(* CODESYS project festo_cpx_api_ec_beckhoff.library
   DefaultNamespace: Festo_CPX_AP_I_EC
   DocFormat: reStructuredText
   Description: FB's for integrating CPX_AP_I_EC_M12 module
   Author: INOSKSR
   Title: Festo_CPX_API_EC_Beckhoff
   Version: 3.5.12.2
   Company: Festo
   Placeholder: Festo_CPX_AP_I_EC

Project tree, tasks and I/O mapping:
  libraries: Tc2_EtherCAT, * (Beckhoff Automation GmbH); Tc2_Standard, * (Beckhoff Automation GmbH); Tc2_System, * (Beckhoff Automation GmbH); Tc3_Module, * (Beckhoff Automation GmbH)
  DUTs/
    function block Restart_Slave [ST]
    data type stModuleDiagData
  ENUMs/
    data type eErrorDescription
    data type eIOLinkAbortCode
    data type eSDOAbortCode
  POUs/
    function block CPXAPI_Diag [ST]
    function block CPXAPI_IOLink_Parameter [ST]
    function block CPXAPI_Parameter [ST]
  Project Information/
    function F_GetCompany [ST]
    function F_GetTitle [ST]
    function F_GetVersion [ST]
  UNIONs/
    data type UDINT_AS_ARRAYOFBYTE
    data type UINT_AS_ARRAYOFBYTE
  Version/
    global variables Global_Version
  VISUs/
    visualisation VISU_CPXAPI_Diag
    visualisation VISU_CPXAPI_IOLinkParameter
    visualisation VISU_CPXAPI_Parameter
  text list GlobalTextList
*)

// DUTs/stModuleDiagData
TYPE stModuleDiagData :
STRUCT
	udiModuleDiagState     : UDINT;
    uiActiveDiagnosisCount : UINT;
	uiSubModule            : UINT;
	uiChannel              : UINT;
	udiDiagnosisCode       : UDINT;
	eErrorDescription      : eErrorDescription;
	xError                 : BOOL;
END_STRUCT
END_TYPE

// ENUMs/eErrorDescription
TYPE eErrorDescription :
(
	NO_ERROR                                              := 0 ,
	OVERVOLTAGE_LOAD_SUPPLY_PS                            := 33619991,
	UNDERVOLTAGE_LOAD_SUPPLY_PL                           := 33620229,
	SWITCH_OFF_LOAD_SUPPLY_PL                             := 33620230,
	OVERVOLTAGE_LOAD_SUPPLY_PL                            := 33620287,
	START_UP_PARAMETER_REJECTED                           := 100663561,
	START_UP_PARAMETER_DEVIATION_IN_LENGTH                := 100663562,
	MODULE_IDENTIFICATION_CHECK_SKIPPED                   := 100663688,
	MODULE_IDENTIFICATION_CHECK_FAILED                    := 100663689,
	DEVICE_ADDRESS_INVALID                                := 134218030,
	INVALID_CYCLE_TIME                                    := 134218130,
	AP_MASTER_LOST                                        := 134283556,
	COMMUNICATION_TO_AP_MODULE_INTERRUPTED                := 134283559,
	OUTPUT_PROCESS_DATA_WATCHDOG_OF_THE_AP_MODULE_EXPIRED := 134283568,
	INPUT_PROCESS_DATA_WATCHDOG_OF_THE_AP_MODULE_EXPIRED  := 134283569,                                   
	OUTPUT_PROCESS_DATA_WATCHDOG_OF_THE_INTERFACE_EXPIRED := 134283570,
	INPUT_PROCESS_DATA_WATCHDOG_OF_THE_INTERFACE_EXPIRED  := 134283571,	
	AP_MASTER_TOGGLE_BIT_ERROR                            := 134283572,
	STATUS_CHANGE_REQUEST                                 := 134480273,
	SYNC_MANAGER_INVALID_ADDRESS                          := 134480275,
	SYNC_MANAGER_INVALID_IO_SIZE                          := 134480276,
	SYNC_MANAGER_INVALID_CONFIGURATION                    := 134480277,
	DC_ACTIVATION_REGISTER_INVALID                        := 134480278,
	SYNC_TYPE_NOT_SUPPORTED                               := 134480279,
	SYSTEM_START                                          := 184549696,
	FIRMWARE_INVALID                                      := 184811703,
	UNSUPPORTED_FULL_DIAGNOSTIC_IMAGE_VERSION             := 185074063,
	UNSUPPORTED_DIAGNOSTIC_VERSION                        := 185074064,
	APDD_INVALID                                          := 185139496,
	START_UP_APDD_INVALID                                 := 185139497,
	INVALID_SLAVEID_OR_COMMUNICATION_ERROR                := 65535
)DWORD;
END_TYPE

// ENUMs/eIOLinkAbortCode
TYPE eIOLinkAbortCode :
(
  NO_ERROR                     := 16#0,
  SERVICE_NOT_AVAILABLE        := 16#8020,
  INDEX_NOT_AVAILABLE          := 16#8011,
  SUB_INDEX_NOT_AVAILABLE      := 16#8012,
  INDEX_NOT_WRITEABLE          := 16#8023 ,
  PARAMETER_VALUE_OUT_OF_RANGE := 16#8030,
  PARAMETER_VALUE_ABOVE_LIMIT  := 16#8031,
  PARAMETER_VALUE_BELOW_LIMIT  := 16#8032,
  PARAMETER_LENGTH_OVERRUN     := 16#8033,
  PARAMETER_LENGTH_UNDERRUN    := 16#8034,
  VENDOR_SPECIFIC              := 16#8181,
  WRONG_SLOT_NUMBER            := 16#703
)DINT;
END_TYPE

// ENUMs/eSDOAbortCode
TYPE eSDOAbortCode :
(
    NO_ERROR                            := 16#0,
	INTERNAL_ERROR                      := 16#1 ,
    NO_REAL_TIME_ERROR                  := 16#2 ,
	PORT_NOT_CONNECTED                  := 16#D,
    GENERAL_DEVICE_ERROR                := 16#700 ,
	SERVICE_NOT_SUPPORTED_BY_SERVER     := 16#701 ,
	INVALID_INDEX_GROUP                 := 16#702 ,
	INVALID_INDEX_OFFSET                := 16#703 , 
	READING_OR_WRITTING_NOT_PERMITTED   := 16#704,
	PARAMETER_SIZE_INCORRECT            := 16#705,
	INVALID_DATA_VALUES                 := 16#706,
	DEVICE_NOT_READY                    := 16#707,
	DEVICE_BUSY                         := 16#708,
	INSUFFICIENT_MEMORY                 := 16#70A,
	INVALID_PARAMETER_VALUES            := 16#70B,
	SYNTAX_ERROR                        := 16#70D
	
	
)DINT;
END_TYPE

// UNIONs/UDINT_AS_ARRAYOFBYTE
TYPE UDINT_AS_ARRAYOFBYTE :
UNION
	dataUDINT: UDINT;
	dataArray : ARRAY[1..4] OF BYTE;
END_UNION
END_TYPE

// UNIONs/UINT_AS_ARRAYOFBYTE
TYPE UINT_AS_ARRAYOFBYTE :
UNION
	dataUINT  : UINT;
	dataArray : ARRAY[1..2] OF BYTE;
END_UNION
END_TYPE

// Version/Global_Version
{attribute 'TcGenerated'}
{attribute 'no-analysis'}
{attribute 'linkalways'}
// This function has been automatically generated from the project information.
VAR_GLOBAL CONSTANT
	{attribute 'const_non_replaced'}
	stLibVersion_Festo_CPX_API_EC_Beckhoff : ST_LibVersion := (iMajor := 3, iMinor := 5, iBuild := 12, iRevision := 2, nFlags := 0, sVersion := '3.5.12.2');
END_VAR

// DUTs/Restart_Slave
FUNCTION_BLOCK Restart_Slave
VAR_INPUT
	xExecute	: 	BOOL;
	sNetId		: 	STRING;
	nSlaveAddr	: 	UINT;
END_VAR
VAR_OUTPUT
	xDone			:	 BOOL;
	xBusy			: 	BOOL;
	xError			: 	BOOL;
	udiError		: 	UDINT;
	stSlaveState	:	Tc2_EtherCAT.ST_EcSlaveState;
END_VAR
VAR
	SetState		: 	FB_EcSetSlaveState;
	GetState		: 	FB_EcGetSlaveState;
	rTrigStart		: 	R_TRIG;
	iStep			: 	INT;
	ReadState		: 	Tc2_EtherCAT.ST_EcSlaveState;
	ExpectedState	: 	UINT := 1;
END_VAR

SetState(sNetId:= sNetId,nSlaveAddr:=nSlaveAddr,tTimeout := T#1S);
GetState(sNetId:= sNetId,nSlaveAddr:=nSlaveAddr,tTimeout := T#1S,state => ReadState);
rTrigStart(CLK := xExecute);

CASE iStep OF
0:
	SetState.bExecute := FALSE;
	GetState.bExecute := FALSE;
	IF rTrigStart.Q THEN
		xBusy := TRUE;
		xError := FALSE;
		xDone := FALSE;
		udiError := 0;
		SetState.reqState := 1;
		ExpectedState := 1;
		iStep := iStep +10;
	END_IF;
	
10:
	SetState.bExecute := TRUE;
	iStep := iStep +10;

20:
	IF NOT SetState.bBusy AND NOT SetState.bError THEN
		SetState.bExecute := FALSE;
		iStep := iStep +10;	
	ELSIF SetState.bError THEN
		udiError := SetState.nErrId;
		iStep := 999;
	END_IF;
	
30:
	GetState.bExecute := TRUE;
	iStep := iStep +10;

40:
	IF NOT GetState.bBusy AND NOT GetState.bError THEN
		GetState.bExecute := FALSE;	
		iStep := iStep +10;
	ELSIF SetState.bError THEN
		udiError := GetState.nErrId;
		iStep := 999;	
	END_IF;
	
50:
	IF ReadState.deviceState = ExpectedState THEN
		SetState.reqState := SHL(SetState.reqState,1);
		ExpectedState := SetState.reqState;
		IF ExpectedState > 8 THEN
			iStep := iStep+10;
		ELSE
			iStep := 10;
		END_IF;
	ELSE
		iStep := 30;
	END_IF;	

60:	
	xBusy := FALSE;
	xError := FALSE;
	xDone := TRUE;
	stSlaveState := ReadState;
	iStep := 0;

999:
	xBusy := FALSE;
	xError := TRUE;
	xDone := FALSE;
	iStep := 0;
	
END_CASE;

END_FUNCTION_BLOCK

// POUs/CPXAPI_Diag
FUNCTION_BLOCK CPXAPI_Diag
VAR_INPUT
	xEnable             : BOOL;              (* TRUE = Start diagnosis continously *)
	sNetId              : STRING;
	uiEthercatAddress   : UINT;              (* Address of the slave device i.e. CPX-AP-I-EC-M12 Module*)
	xRestart            : BOOL;              (* Change Machine State in order INIT, PREOP, SAFE and OPERATIONAL*)
END_VAR

VAR_OUTPUT
	xActive						 : BOOL;	 (*  Diagnosis FB Active *)
	xError                       : BOOL;     (*  Error exists during diagnosis *)
	uiActiveModules              : UINT;     (*  Number of Active modules connected to CPX-AP-I-EC-M12*)
	uiNumberOfActiveErrors       : UINT;     (* Number of Modules with active errors*)
	uiModuleNo                   : UINT;     (* Module with latest diagnostics*)
	aModuleDiagnosticData        : ARRAY[1..150] OF stModuleDiagData ;
END_VAR
VAR
	ReadModuleCount			:	FB_EcCoESdoReadEx;
	ModuleDiagnosis			:	FB_EcCoESdoReadEx;
	aModuleCount			:	ARRAY[1..150] OF UDINT;
	ModuleDiagnosisData		:	ARRAY[1..150] OF BYTE;
	R_Trig_Exec         	:	R_TRIG;
	F_Trig_Exec				:	F_TRIG;
	iStep					:	INT;
	Delay					:	TON;
	xDelay					:	BOOL;
	DelayUpdate				:	TON;
	xDelayUpdate			:	BOOL;
	i						:	INT;
	k						:	INT;
	Acknowledge_Trig		:	R_TRIG;
	Restart_RTrig         	:	R_TRIG;
	iRestart				:	INT;
	Restart_FTrig			:	F_TRIG;
	diActualIndex         	:	DINT;
	iCurrentModuleDiag    	: 	INT;
	DiagCode				:	DWORD;
	ModuleDiagState			:	UDINT_AS_ARRAYOFBYTE;
	DiagnosisCode			:	UDINT_AS_ARRAYOFBYTE;
	SubModule				: 	UINT_AS_ARRAYOFBYTE;
	Channel					: 	UINT_AS_ARRAYOFBYTE;
	NumberOfActiveModules	: 	UINT_AS_ARRAYOFBYTE;
	j                     	: 	INT;
	l                     	: 	INT;
	tempmodules           	: 	ARRAY[1..150] OF INT;
	DelayRequestSlave		:	TON;
	xDelayRequestSlave		:	BOOL;
	iActive					:	INT;
	F_Trig_Active			:	F_TRIG;
	ActiveOff				:	TON;
	xActiveOff				:	BOOL;
	DelayON					:	TON;
	xDelayON				:	BOOL;
	iRestartCount			:	INT;
	iCurrentRestartCount	:	INT;
	SlaveChangeState		: 	Restart_Slave;
	GetSlaveState			:	FB_EcGetSlaveState;
END_VAR

R_Trig_Exec( CLK := xEnable);
F_Trig_Exec( CLK := xEnable);
Restart_RTrig( CLK := xRestart);
Restart_FTrig( CLK := xRestart);
F_Trig_Active( CLK := xActive);

Delay ( IN := xDelay, PT:= T#100MS);
DelayUpdate ( IN := xDelayUpdate, PT:= T#50MS);

ActiveOff ( IN := xActiveOff, PT:= T#500MS);

DelayON ( IN := xDelayON, PT := T#1S );

DelayRequestSlave ( IN := xDelayRequestSlave, PT:= T#50MS);

IF Restart_RTrig.Q THEN
	iRestartCount	:=	iRestartCount + 1;
END_IF

SlaveChangeState(
	xExecute		:= 	,
	sNetID			:=	sNetId , 
	nSlaveAddr		:=	uiEthercatAddress,
	xDone			=>	,
	xBusy			=>	,
	xError			=>	,
	udiError		=>	,
	stSlaveState	=>	);

GetSlaveState(
	sNetId			:=	sNetId , 
	nSlaveAddr		:=	uiEthercatAddress,
	bExecute		:=	,
	tTimeout		:=	T#1S,
	bBusy			=>	,
	bError			=>	,
	state			=>	);	
	
ReadModuleCount(
	sNetId			:=	sNetId , 
	nSlaveAddr		:=	uiEthercatAddress,   
	nSubIndex		:= 	1, 
	nIndex			:= 	16#F050, 
	pDstBuf			:= 	ADR(aModuleCount), 
	cbBufLen		:= 	SIZEOF(aModuleCount), 
	bExecute		:= 	, 
	tTimeout		:= 	T#1000MS, 
	bCompleteAccess	:= 	TRUE, 
	bBusy			=> 	, 
	bError			=> 	, 
	nErrId			=> 	, 
	cbRead			=> 	);

ModuleDiagnosis(
	sNetId			:= 	sNetId, 
	nSlaveAddr		:=	uiEthercatAddress,  
	nSubIndex		:= 	1, 
	nIndex			:=	TO_WORD(diActualIndex) , 
	pDstBuf			:= 	ADR(ModuleDiagnosisData), 
	cbBufLen		:= 	SIZEOF(ModuleDiagnosisData), 
	bExecute		:= 	, 
	tTimeout		:= 	, 
	bCompleteAccess	:= 	TRUE, 
	bBusy			=> 	, 
	bError			=> 	, 
	nErrId			=> 	, 
	cbRead			=> 	);
	
IF Restart_FTrig.Q OR F_Trig_Exec.Q THEN
	iRestart := 0;
	SlaveChangeState.xExecute  := FALSE;
END_IF

CASE iRestart OF
	0:
		SlaveChangeState.xExecute := FALSE;
		iRestart := iRestart + 5;
		
	5:
		IF xEnable THEN
	      iRestart := iRestart + 5;
		END_IF
		
	10:
		IF Restart_RTrig.Q THEN
			xActive := FALSE;
		   	iRestart := iRestart + 10;
		END_IF
		
	20:
		SlaveChangeState.xExecute := TRUE;
		iRestart := iRestart + 10;
	
	30:
		IF SlaveChangeState.xDone THEN
			SlaveChangeState.xExecute := FALSE;
			iRestart := iRestart + 10;
		END_IF
		
	40:
        IF Restart_FTrig.Q THEN
			iRestart := 0;
		END_IF
		
END_CASE

CASE iActive OF
	0:
		GetSlaveState.bExecute := FALSE;
	 	xDelayON := FALSE;
		xDelayRequestSlave := FALSE;
     	iActive := iActive + 10;
		
	10:
		IF xEnable THEN
			GetSlaveState.bExecute := TRUE;
			xDelayRequestSlave := TRUE;
         	iActive := iActive + 5;	
	 	END_IF
		
	15:
		IF DelayRequestSlave.Q THEN
			xDelayRequestSlave := FALSE;
			iActive := iActive + 5;
	 	END_IF
		
	20:
		IF NOT GetSlaveState.bBusy AND NOT GetSlaveState.bError THEN
			iActive := iActive + 10;
		ELSE
			iActive := 0;
		END_IF
	
	30:
		IF GetSlaveState.state.deviceState = 8 THEN
			GetSlaveState.bExecute := FALSE;
			iActive := iActive + 10;
		ELSIF GetSlaveState.state.linkState <> 0 THEN
			xActive	:=	FALSE;
			iActive := 	50;
		ELSE
			GetSlaveState.bExecute := FALSE;
			iActive := 10;
		END_IF
		
	40:
		IF xEnable AND GetSlaveState.state.linkState = 0 THEN
			xActive	:=	TRUE;
			iCurrentRestartCount := iRestartCount;
			iActive := iActive + 5;
		ELSE
			xActive	:=	FALSE;
			iActive := 	50;
		END_IF
		
	45:
		xDelayON := TRUE;
		IF DelayON.Q THEN
			xDelayON := FALSE;
			iActive := 10;
		END_IF
		
	50:
		IF NOT xActive THEN
			GetSlaveState.bExecute := FALSE;
			xActiveOff := TRUE;
			uiActiveModules := 0;
			iStep := 0;
			iActive := iActive + 10;
		END_IF
		
	60:
		IF ActiveOff.Q THEN
			xActiveOff := FALSE;
			xDelayON := FALSE;
			iActive := iActive + 10;
		END_IF
	
	70:
		IF iRestartCount = iCurrentRestartCount THEN
			SlaveChangeState.xExecute := TRUE;
			iActive := iActive + 5;
		ELSE
			iActive := 10;
		END_IF
	
	75:
		xDelayRequestSlave := TRUE;
		IF DelayRequestSlave.Q THEN
			xDelayRequestSlave := FALSE;
			iActive := iActive + 5;
		END_IF
		
	80:
		IF SlaveChangeState.xDone THEN
			SlaveChangeState.xExecute := FALSE;
			iActive := iActive + 10;
		ELSIF NOT SlaveChangeState.xBusy THEN
			SlaveChangeState.xExecute := FALSE;
			iActive := 50;
		END_IF
			
	90:
		IF SlaveChangeState.stSlaveState.deviceState = 8 THEN
			iActive := 10;
		END_IF
END_CASE

CASE iStep OF

 	0:
     	ModuleDiagnosis.bExecute := FALSE;
     	ReadModuleCount.bExecute := FALSE;
		iStep := iStep + 10;

	10:
		IF xEnable AND xActive THEN
         	iStep := iStep + 10;
		END_IF
	
	20:
     	ReadModuleCount.bExecute := TRUE;
	 	xDelayUpdate := TRUE;
		iStep := iStep + 5;
	 
	25:
		IF DelayUpdate.Q THEN
			xDelayUpdate := FALSE;
			iStep := iStep + 5;
	 	END_IF
	
	30:
     	IF NOT ReadModuleCount.bBusy AND NOT ReadModuleCount.bError THEN
			iStep := iStep +10;
		ELSIF ReadModuleCount.bError THEN
			ReadModuleCount.bExecute := FALSE;
			iStep := 999;
		END_IF
	 
	40:
		FOR i:= 1 TO 150 DO
			IF aModuleCount[i] <> 0 THEN
				uiActiveModules := uiActiveModules + 1;
			END_IF
		END_FOR
		ReadModuleCount.bExecute := FALSE;
		iStep := iStep + 5;
		
	45:
		IF uiActiveModules > 0 THEN
			iStep := iStep + 5;
		ELSE
			iStep := 20;
		END_IF
	
	50:
		IF iCurrentModuleDiag = TO_INT(uiActiveModules) THEN
			iStep := 110;
		ELSE
			iStep := iStep + 10;
		END_IF
	
	60:
		diActualIndex := 16#A000 + iCurrentModuleDiag;
		ModuleDiagnosis.bExecute := TRUE;
		xDelayUpdate := TRUE;
		iStep := iStep + 5;
		 
	65:
		IF DelayUpdate.Q THEN
	    	xDelayUpdate := FALSE;
	    	iStep := iStep + 5;
	 	END_IF
	 
	70:
		IF NOT ModuleDiagnosis.bBusy AND NOT ModuleDiagnosis.bError THEN
			iStep := iStep + 10;
		ELSIF ModuleDiagnosis.bError THEN
			ModuleDiagnosis.bExecute := FALSE;
			iStep := 999;
		END_IF
		
	80: 
		iCurrentModuleDiag := iCurrentModuleDiag + 1;
		iStep := iStep + 10;
	90:
		// Module Diag State
		ModuleDiagState.dataArray[1] := ModuleDiagnosisData[1];
		ModuleDiagState.dataArray[2] := ModuleDiagnosisData[2];
		ModuleDiagState.dataArray[3] := ModuleDiagnosisData[3];
		ModuleDiagState.dataArray[4] := ModuleDiagnosisData[4];
		
		// Number of Active Modules
		NumberOfActiveModules.dataArray[1] := ModuleDiagnosisData[5];
		NumberOfActiveModules.dataArray[2] := ModuleDiagnosisData[6];
		
		// Sub Module
		SubModule.dataArray[1] := ModuleDiagnosisData[7];
		SubModule.dataArray[2] := ModuleDiagnosisData[8];
		
		// Channel
		Channel.dataArray[1] := ModuleDiagnosisData[9];
		Channel.dataArray[2] := ModuleDiagnosisData[10];
		
		 // Diagnosis Code
		DiagnosisCode.dataArray[1] := ModuleDiagnosisData[11];
		DiagnosisCode.dataArray[2] := ModuleDiagnosisData[12];
		DiagnosisCode.dataArray[3] := ModuleDiagnosisData[13];
		DiagnosisCode.dataArray[4] := ModuleDiagnosisData[14];
	
		iStep := iStep + 10;
				
	100:
		aModuleDiagnosticData[iCurrentModuleDiag].udiModuleDiagState     := ModuleDiagState.dataUDINT;
		aModuleDiagnosticData[iCurrentModuleDiag].uiActiveDiagnosisCount := NumberOfActiveModules.dataUINT;
		aModuleDiagnosticData[iCurrentModuleDiag].uiSubModule            := SubModule.dataUINT;
		aModuleDiagnosticData[iCurrentModuleDiag].uiChannel              := Channel.dataUINT;
		aModuleDiagnosticData[iCurrentModuleDiag].udiDiagnosisCode       := DiagnosisCode.dataUDINT;
		aModuleDiagnosticData[iCurrentModuleDiag].eErrorDescription      := aModuleDiagnosticData[iCurrentModuleDiag].udiDiagnosisCode;
		ModuleDiagnosis.bExecute := FALSE;
		iStep := 50;
		
	110:
		FOR j:= 1 TO TO_INT(uiActiveModules) DO
			IF j <> TO_INT(uiActiveModules + 1 ) THEN
				IF aModuleDiagnosticData[j].udiModuleDiagState <> 1 AND NOT aModuleDiagnosticData[j].xError THEN
					aModuleDiagnosticData[j].xError := TRUE;
					uiNumberOfActiveErrors := uiNumberOfActiveErrors + 1;
					uiModuleNo := TO_UINT(j);
				ELSIF aModuleDiagnosticData[j].udiModuleDiagState = 1 AND aModuleDiagnosticData[j].xError AND uiNumberOfActiveErrors > 0 THEN
					uiNumberOfActiveErrors := uiNumberOfActiveErrors - 1;
				 	aModuleDiagnosticData[j].xError := FALSE;
				END_IF
			END_IF
		END_FOR	 
		 iStep := iStep + 10;
		 
	120:
		IF uiNumberOfActiveErrors > 0 THEN
			iStep := 999;
		ELSE
			xError := FALSE;
			uiModuleNo := 0;
			iStep := 130;
		END_IF

	130:
		xDelay := TRUE;
		iStep := iStep + 10;
		   
	140:
		IF Delay.Q THEN
		   iCurrentModuleDiag := 0;
		   xDelay := FALSE;
		   iStep := 50;
		END_IF
		
	999:
		xError := TRUE;
		iCurrentModuleDiag := 0;
		iStep := 50;
END_CASE

IF F_Trig_Exec.Q THEN
	iActive := 0;
	xActive := FALSE;
	xDelayUpdate := FALSE;
	xDelay := FALSE;
	ReadModuleCount.bExecute := FALSE;
	ModuleDiagnosis.bExecute := FALSE;
	xError := FALSE;
	iCurrentModuleDiag := 0;
	uiActiveModules := 0;
	uiModuleNo := 0;
	uiNumberOfActiveErrors := 0;
	iRestartCount := 0;
	iCurrentRestartCount := 0;
	FOR k:= 1 TO 150 DO
		aModuleDiagnosticData[k].udiDiagnosisCode := 0;
		aModuleDiagnosticData[k].udiModuleDiagState := 0;
		aModuleDiagnosticData[k].uiActiveDiagnosisCount :=0;
		aModuleDiagnosticData[k].uiChannel := 0;
		aModuleDiagnosticData[k].uiSubModule := 0;
		aModuleDiagnosticData[k].eErrorDescription := 0;
		aModuleDiagnosticData[k].xError := FALSE;
	END_FOR
	iStep := 0;
END_IF

END_FUNCTION_BLOCK

// POUs/CPXAPI_IOLink_Parameter
FUNCTION_BLOCK CPXAPI_IOLink_Parameter
VAR_INPUT
	xExecute            : BOOL;               (* TRUE = Start Parameter Read or Write operation*)
	sNetId              : STRING;
	uiEthercatAddress   : UINT;               (* Address of the slave device i.e. CPX-AP-I-EC-M12 Module*)
	uiSlotNumber        : UINT;               (* Slot number where the IO Link master CPX-AP-I-4IOL-M12 module is connected*)
	usiPort             : USINT;              (* Port of the CPX-AP-I-4IOL-M12 module where IO link device is connected *)
	uiIndex             : UINT;               (* Index of the IO Link device parameter to be read/write*)
	usiSubIndex         : USINT;              (* Sub Index of the IO Link device parameter to be read/write*)
	pData	            : POINTER TO BYTE;    (* Pointer to the variable which holds the data to be read or written*)
	uiDataLength        : UINT;               (* Number of bytes of data to be  written*)
	xWrite          : BOOL;               	  (* TRUE = Parameter write, FALSE = Parameter Read*)
	xIsString           : BOOL;               (* TRUE if the parameter is of STRING data type*)
END_VAR
VAR_OUTPUT
	xDone               : BOOL;               (* Parameter Read/Write is completed successfuly*)
	xBusy               : BOOL;               (* Parameter Read /Write is under progress *)
	xError              : BOOL;               (* TRUE = Error when doing Parameter Read or Write*)
	udiErrorCode        : UDINT;              (* Error code generate during Parameter read or write*)
	eErrorDescription   : eIOLinkAbortCode;      (* Error Code description *)
	udiReadDataLength    : UDINT;              (* Number of bytes of data read *)
END_VAR
	

VAR
   	EcCoESdoWritePort: FB_EcCoESdoWriteEx;
	EcCoESdoWriteIndex: FB_EcCoESdoWriteEx;
	EcCoESdoWriteSubIndex: FB_EcCoESdoWriteEx;
	EcCoESdoWriteDataLength: FB_EcCoESdoWriteEx;
	EcCoESdoWriteDirection: FB_EcCoESdoWriteEx;
	EcCoESdoReadISDUCError: FB_EcCoESdoReadEx;
	EcCoESdoReadDataArray: FB_EcCoESdoReadEx;
	EcCoESdoWriteDataArray: FB_EcCoESdoWriteEx;
	EcCoESdoReadDataLength: FB_EcCoESdoReadEx;
	aECATParameterReadData  : ARRAY [0..237] OF BYTE;
	aECATParameterWriteData : ARRAY [0..237] OF BYTE;
	pDestination            : ARRAY [0..237] OF POINTER TO  BYTE;
	wActualIndex            : WORD;
	usiDirection            : USINT;
	udiErrorCodePort        : UDINT;
	udiErrorCodeIndex       : UDINT;	
    udiErrorCodeSubIndex    : UDINT;
	udiErrorCodeLength      : UDINT;
	udiErrorCodeDirection   : UDINT;
	udiErrorCodeISDU        : UDINT;
	udiErrorCodeReadParam   : UDINT;
	udiErrorCodeWriteParam  : UDINT;
	R_Trig_Exec             : R_TRIG;
	F_Trig_Exec             : F_TRIG;
	iStep                   : INT;
	iByteCount              : UDINT;
	iByteCountWrite         : UINT;
	i                       : UDINT;
	j                       : UINT;
	k                       : UINT;
	bActualSubIndex         : BYTE;
	uiLength                : UINT;
	uiData                  : UINT;
	wParameterValue         : DWORD;
	DelayRead               : TON;
	xDelayRead              : BOOL;
	uiISDUErrorTemp         : UDINT;
	DONE_RTRIG              : R_TRIG;
    LengthRead              : UDINT;

END_VAR

R_Trig_Exec( CLK := xExecute);
F_Trig_Exec( CLK := xExecute);
DONE_RTRIG ( CLK := xDone);

wActualIndex := 8704 + ( uiSlotNumber - 1);  
usiDirection.0 :=  xWrite;

 wParameterValue := TO_DWORD(aECATParameterReadData[0]) + SHL(TO_DWORD(aECATParameterReadData[1]),16) + SHL(TO_DWORD(aECATParameterReadData[2]),16)+ SHL(TO_DWORD(aECATParameterReadData[3]),16);  
DelayRead ( IN := xDelayRead, PT:= T#200MS);

//Parameter Read when Data Type is STRING.
IF DONE_RTRIG.Q AND NOT xWrite AND  xIsString  THEN
	iByteCount := udiReadDataLength;
	pDestination[0] := pData;
    FOR i:= 0 TO iByteCount -1 DO
	   pDestination[i]  := pDestination[0]+i;
	   pDestination[i]^ := aECATParameterReadData[i];
    END_FOR
END_IF

//Parameter Read when Data Type is not STRING.
IF DONE_RTRIG.Q AND NOT xWrite AND NOT xIsString THEN
	iByteCount := udiReadDataLength;
	pDestination[0] := pData;
    FOR i:= 0 TO iByteCount -1 DO
	   pDestination[i]  := pDestination[0]+i;
	   pDestination[i]^ := aECATParameterReadData[iByteCount-1-i];
    END_FOR
END_IF

//Parameter write when Data Type is STRING.
IF xWrite AND uiDataLength > 0 AND  xIsString THEN
	iByteCountWrite := uiDataLength;
	pDestination[0] := pData;
	FOR j:= 0 TO iByteCountWrite -1 DO
	   pDestination[j] := pDestination[0]+j;
	   aECATParameterWriteData[j]  := pDestination[j]^;
	END_FOR
END_IF

//Parameter write when Data Type is not STRING.
IF xWrite AND uiDataLength > 0 AND NOT xIsString THEN
	iByteCountWrite := uiDataLength;
	pDestination[0] := pData;
	FOR j:= 0 TO iByteCountWrite -1 DO
	   pDestination[j] := pDestination[0]+j;
	   aECATParameterWriteData[iByteCountWrite-1-j]  := pDestination[j]^;
	END_FOR
END_IF


// Write Port Number 
EcCoESdoWritePort (
	sNetId:= sNetId, 
	nSlaveAddr:= uiEthercatAddress, 
	nSubIndex:= 2, 
	nIndex:= wActualIndex, 
	pSrcBuf:= ADR(usiPort), 
	cbBufLen:= 1, 
	bExecute:= , 
	tTimeout:= T#1000MS, 
	bCompleteAccess:= FALSE, 
	bBusy=> , 
	bError=> , 
	nErrId=> udiErrorCodePort);

// Write Index 	
EcCoESdoWriteIndex      (
	sNetId:= sNetId, 
	nSlaveAddr:= uiEthercatAddress, 
	nSubIndex:= 3, 
	nIndex:= wActualIndex, 
	pSrcBuf:= ADR(uiIndex), 
	cbBufLen:= 2, 
	bExecute:= , 
	tTimeout:=T#1000MS , 
	bCompleteAccess:= FALSE, 
	bBusy=> , 
	bError=> , 
	nErrId=> udiErrorCodeIndex);
	
	// Write Sub Index
EcCoESdoWriteSubIndex   (
	sNetId:= sNetId, 
	nSlaveAddr:= uiEthercatAddress, 
	nSubIndex:= 4, 
	nIndex:= wActualIndex, 
	pSrcBuf:= ADR(usiSubIndex), 
	cbBufLen:= 1, 
	bExecute:= , 
	tTimeout:=T#1000MS , 
	bCompleteAccess:= FALSE, 
	bBusy=> , 
	bError=> , 
	nErrId=> udiErrorCodeSubIndex);
	
	// Write Data Length
EcCoESdoWriteDataLength (
	sNetId:= sNetId, 
	nSlaveAddr:= uiEthercatAddress, 
	nSubIndex:= 6, 
	nIndex:= wActualIndex, 
	pSrcBuf:= ADR(uiDataLength), 
	cbBufLen:= 1, 
	bExecute:= , 
	tTimeout:=T#1000MS , 
	bCompleteAccess:= FALSE, 
	bBusy=> , 
	bError=> , 
	nErrId=> udiErrorCodeLength);
	
	//Write Direction
EcCoESdoWriteDirection  (
	sNetId:= sNetId, 
	nSlaveAddr:= uiEthercatAddress, 
	nSubIndex:= 1, 
	nIndex:= wActualIndex, 
	pSrcBuf:= ADR(usiDirection), 
	cbBufLen:= 1, 
	bExecute:= , 
	tTimeout:= T#1000MS, 
	bCompleteAccess:= FALSE, 
	bBusy=> , 
	bError=> , 
	nErrId=> udiErrorCodeDirection);
	
	//Read ISDU Error
EcCoESdoReadISDUCError  (
	sNetId:= sNetId, 
	nSlaveAddr:= uiEthercatAddress, 
	nSubIndex:= 5, 
	nIndex:= wActualIndex, 
	pDstBuf:= ADR(uiISDUErrorTemp), 
	cbBufLen:= 2, 
	bExecute:= , 
	tTimeout:= T#1000MS, 
	bCompleteAccess:= FALSE, 
	bBusy=> , 
	bError=> , 
	nErrId=>udiErrorCodeISDU , 
	cbRead=> );

	// Read Parameter Data
EcCoESdoReadDataArray   (
	sNetId:= sNetId, 
	nSlaveAddr:= uiEthercatAddress, 
	nSubIndex:= 7, 
	nIndex:= wActualIndex, 
	pDstBuf:= ADR(aECATParameterReadData), 
	cbBufLen:= SIZEOF(aECATParameterReadData), 
	bExecute:= , 
	tTimeout:= T#1000MS, 
	bCompleteAccess:= FALSE, 
	bBusy=> , 
	bError=> , 
	nErrId=>udiErrorCodeReadParam , 
	cbRead=> );
	
	
	//Write Parameter Data

	EcCoESdoWriteDataArray  (
	sNetId:= sNetId, 
	nSlaveAddr:= uiEthercatAddress, 
	nSubIndex:= 7, 
	nIndex:= wActualIndex, 
	pSrcBuf:= ADR(aECATParameterWriteData), 
	cbBufLen:= SIZEOF(aECATParameterWriteData), 
	bExecute:= , 
	tTimeout:= T#1000MS, 
	bCompleteAccess:= FALSE, 
	bBusy=> , 
	bError=> , 
	nErrId=> udiErrorCodeWriteParam);
	
	EcCoESdoReadDataLength(
	sNetId:= sNetId, 
	nSlaveAddr:= uiEthercatAddress, 
	nSubIndex:= 6, 
	nIndex:= wActualIndex, 
	pDstBuf:= ADR(LengthRead), 
	cbBufLen:= 1, 
	bExecute:= , 
	tTimeout:= T#1000MS, 
	bCompleteAccess:= FALSE, 
	bBusy=> , 
	bError=> , 
	nErrId=> , 
	cbRead=> );
	
CASE iStep OF
	0:
	FOR k := 0 TO 237 DO
		aECATParameterReadData[k] := 0;
		aECATParameterWriteData[k] := 0;
		pDestination[k]:= 0;
	END_FOR
	 istep := istep + 10;
	 
	10:
	   
	   IF R_TRIG_Exec.Q  THEN
		   iStep := 20;
	   END_IF;
	   
	   // Port Number
	20:
	    EcCoESdoWritePort.bExecute := TRUE;
		xDelayRead := TRUE;
        istep := istep + 10;  
		
    30:
	      IF DelayRead.Q THEN
			xDelayRead := FALSE;
			iStep := iStep + 10;
		  END_IF;
	40:
	    IF NOT EcCoESdoWritePort.bError THEN
		    EcCoESdoWritePort.bExecute := FALSE;
			iStep := iStep + 10;
	    ELSE
			udiErrorCode := udiErrorCodePort;
		    eErrorDescription := TO_DINT(udiErrorCode);
			xError := TRUE;
		    EcCoESdoWritePort.bExecute := FALSE;
			iStep := 999;
		END_IF;
		
		// Index
	50:
	   
		EcCoESdoWriteIndex.bExecute := TRUE;
        istep := istep + 10; 
    60:
			iStep := iStep + 10;
	70:
	    IF NOT EcCoESdoWriteIndex.bError THEN
		    EcCoESdoWriteIndex.bExecute := FALSE;
			iStep := iStep + 10;
	    ELSE
			udiErrorCode := udiErrorCodeIndex;
			eErrorDescription := TO_DINT(udiErrorCode);
		    EcCoESdoWriteIndex.bExecute := FALSE;			
			xError := TRUE;
			iStep := 999;
		END_IF;
	
    // Sub Index	
	80:
	   
		EcCoESdoWriteSubIndex.bExecute := TRUE;
        istep := istep + 10;
    90:
			iStep := iStep + 10;
  	100:
	    IF NOT EcCoESdoWriteSubIndex.bError THEN
		    EcCoESdoWriteSubIndex.bExecute := FALSE;
			iStep := iStep + 10;
	    ELSE
			udiErrorCode := udiErrorCodeSubIndex;
			eErrorDescription := TO_DINT(udiErrorCode);
		    EcCoESdoWriteSubIndex.bExecute := FALSE;			
			xError := TRUE;
			iStep := 999;
		END_IF;
		
   110:
       	IF NOT xWrite  THEN;
           istep := 180; 
		ELSE
			iStep := iStep + 10;
        END_IF;   		
	
    // Length of data	
	120:
	   
		EcCoESdoWriteDataLength.bExecute := TRUE;
        istep := istep + 10; 
    130:
			iStep := iStep + 10;
 	140:
	    IF NOT EcCoESdoWriteDataLength.bError THEN
		    EcCoESdoWriteDataLength.bExecute := FALSE;
			iStep := iStep + 10;
	    ELSE
			udiErrorCode := udiErrorCodeLength;
			eErrorDescription := TO_DINT(udiErrorCode);
		    EcCoESdoWriteDataLength.bExecute := FALSE;		
			xError := TRUE;
			iStep := 999;			
		END_IF;
		
    150 :
	     IF xWrite THEN
			 iStep := iStep + 10;
		 ELSE
			 iStep := 180;
		 END_IF	
			
		  // Write Parameter Data
	160:
	   
		EcCoESdoWriteDataArray.bExecute := TRUE;
		xDelayRead := TRUE;
        istep := istep + 5; 
		
    165:
	     IF DelayRead.Q THEN
			xDelayRead := FALSE; 
			istep := istep + 5; 
		 END_IF
  
	170:
	    IF NOT EcCoESdoWriteDataArray.bError THEN
		    EcCoESdoWriteDataArray.bExecute := FALSE;
			iStep := iStep + 10;
	    ELSE
			udiErrorCode := udiErrorCodeWriteParam;
			eErrorDescription := TO_DINT(udiErrorCode);
			EcCoESdoWriteDataArray.bExecute := FALSE;
			xError := TRUE;
			iStep := 999;
	    END_IF;			
	
		
   // Direction	
	180:
	   
		EcCoESdoWriteDirection.bExecute := TRUE;
        istep := istep + 10; 

	190:
	    IF NOT EcCoESdoWriteDirection.bError THEN
		    EcCoESdoWriteDirection.bExecute := FALSE;
			xDelayRead:= FALSE;
			iStep := iStep + 10;
	    ELSE
			udiErrorCode := udiErrorCodeDirection;
		    eErrorDescription := TO_DINT(udiErrorCode);
		    EcCoESdoWriteDirection.bExecute := FALSE;			
			xError := TRUE;
			iStep := istep + 10;
	    END_IF;			


   // Read ISDU Error	
	200:
	 	EcCoESdoReadISDUCError.bExecute := TRUE;
		xDelayRead := TRUE;
        istep := istep + 10;  
    210:
	    IF DelayRead.Q THEN
			xDelayRead := FALSE;
			iStep := iStep + 10;
	    END_IF;
 
	220:
	    IF uiISDUErrorTemp = 0 THEN
		    EcCoESdoReadISDUCError.bExecute := FALSE;
			iStep := iStep + 10;
	    ELSE
			udiErrorCode := uiISDUErrorTemp;
		    EcCoESdoReadISDUCError.bExecute := FALSE;
			xError := TRUE;
			iStep := 9999;
	    END_IF;	
		
   	230:
	 	IF xWrite  THEN;	
           istep := 1000; 
		ELSE
		 istep := iStep + 10;
        END_IF;   
		
		  // Read Parameter Data
	240:
	   
		EcCoESdoReadDataArray.bExecute := TRUE;
		xDelayRead := TRUE;
        istep := istep + 10;   
		
 	250:
	     IF DelayRead.Q THEN
			 xDelayRead := FALSE;
			 iStep := iStep + 10;
		 END_IF
			
			
	260:
	    IF NOT EcCoESdoReadDataArray.bError THEN
		    EcCoESdoReadDataArray.bExecute := FALSE;
			iStep := iStep + 10;
	    ELSE
			udiErrorCode := udiErrorCodeReadParam;
		    eErrorDescription := TO_DINT(udiErrorCode);
		    EcCoESdoReadDataArray.bExecute := FALSE;			
			xError := TRUE;
			iStep := 999;
	    END_IF;	
		
    270:
        EcCoESdoReadDataLength.bExecute := TRUE;
		xDelayRead := TRUE;
        iStep := iStep + 10;

    280:
	    IF DelayRead.Q THEN
			 xDelayRead := FALSE;
			 udiReadDataLength := LengthRead;
			 iStep := iStep + 10;
		 END_IF
	     
	
	290:
	    IF udiReadDataLength > 0 THEN
		   istep := 1000;
	    ELSE
		   EcCoESdoReadDataLength.bExecute := FALSE;
		   iStep := 270;
		END_IF
	
	  	
	9999:
	    udiErrorCode:= uiISDUErrorTemp;
		eErrorDescription := TO_DINT(udiErrorCode);
	   IF NOT xExecute THEN
		   istep := 0;
	   END_IF;		  
	   
	999:
		
	   IF NOT xExecute THEN
		   istep := 0;
	   END_IF;		  

    1000:
	  xDone := TRUE;
	  EcCoESdoReadDataLength.bExecute := FALSE;
	  IF NOT xExecute THEN
		  istep := 0;
	   END_IF;		  	      
	  
END_CASE;



IF F_TRIG_Exec.Q THEN
	iStep :=0;
	xDone := FALSE;
	xBusy := FALSE;
	xError := FALSE;
	udiErrorCode := 0;
	eErrorDescription := 0;
	udiReadDataLength := 0;
END_IF;

END_FUNCTION_BLOCK

// POUs/CPXAPI_Parameter
FUNCTION_BLOCK CPXAPI_Parameter
VAR_INPUT
	xExecute            : BOOL;                  (* TRUE = Start Parameter Read or Write operation*)
	sNetId              : STRING;
	uiEthercatAddress   : UINT;                  (* Address of the slave device i.e. CPX-AP-I-EC-M12 Module*)
	wIndex              : WORD;                  (* CoE Index of the CPX-AP-I device parameter to be read/write*)
	bySubIndex          : BYTE;                  (* CoE Sub Index of the CPX-AP-I device parameter to be read/write*)
	pData	            : POINTER TO BYTE;       (* Pointer to the variable which holds the data to be read or written*)
	uiDataLength        : UINT;                  (* Number of bytes of data to be  written*)
	xWrite          : BOOL;                  	 (* TRUE = Parameter write, FALSE = Parameter Read*)
END_VAR
VAR_OUTPUT
	xDone               : BOOL;                  (* Parameter Read/Write is completed successfuly*)
	xBusy               : BOOL;                  (* Parameter Read /Write is under progress *)
	xError              : BOOL;                  (* TRUE = Error when doing Parameter Read or Write*)
	udiErrorCode        : UDINT;                 (* Error code generate during Parameter read or write*)
	eErrorDescription   : eSDOAbortCode;         (* Error Code description *)
	udiReadDataLength   : UDINT;                 (* Number of bytes of data read *)
END_VAR
VAR
	EcCoESdoWriteEx: FB_EcCoESdoWriteEx;
	EcCoESdoReadEx: FB_EcCoESdoReadEx;
	aECATParameterReadData  : ARRAY [0..100] OF BYTE;
	aECATParameterWriteData : ARRAY [0..100] OF BYTE;
	pDestination            : ARRAY [0..100] OF POINTER TO  BYTE;
	wActualIndex            : WORD;
	R_Trig_Exec             : R_TRIG;
	F_Trig_Exec             : F_TRIG;
	iStep                   : INT;
	iByteCount              : UDINT;
	iByteCountWrite         : UINT;
	i                       : UDINT;
	j                       : UINT;
	k                       : UINT;
	DelayWrite              : TON;
	xDelayWrite             : BOOL;
	DelayRead               : TON;
	xDelayRead              : BOOL;
	udiAbort                : UDINT;
	Done_TRIG               : R_TRIG;

END_VAR

R_Trig_Exec( CLK := xExecute);
F_Trig_Exec( CLK := xExecute);
Done_TRIG  ( CLK := xDone);

DelayWrite ( IN := xDelayWrite, PT:= T#500MS);
DelayRead ( IN := xDelayRead, PT:= T#500MS);

wActualIndex := wIndex ;

IF Done_TRIG.Q AND NOT xWrite  THEN
	iByteCount := udiReadDataLength;
	pDestination[0] := pData;
    FOR i:= 0 TO iByteCount -1 DO
	   pDestination[i]  := pDestination[0]+i;
	   pDestination[i]^ := aECATParameterReadData[i];
    END_FOR
END_IF

IF xWrite AND uiDataLength > 0 THEN
	iByteCountWrite := uiDataLength;
	pDestination[0] := pData;
	FOR j:= 0 TO iByteCountWrite -1 DO
	   pDestination[j] := pDestination[0]+j;
	   aECATParameterWriteData[j]  := pDestination[j]^;
	END_FOR
END_IF


EcCoESdoWriteEx(
	sNetId:= sNetId, 
	nSlaveAddr:= uiEthercatAddress, 
	nSubIndex:= bySubIndex, 
	nIndex:= wIndex, 
	pSrcBuf:= ADR(aECATParameterWriteData), 
	cbBufLen:= uiDataLength, 
	bExecute:= , 
	tTimeout:= T#1000MS, 
	bCompleteAccess:= FALSE, 
	bBusy=> xBusy, 
	bError=> , 
	nErrId=> );
	
EcCoESdoReadEx(
	sNetId:= sNetId, 
	nSlaveAddr:=uiEthercatAddress , 
	nSubIndex:=bySubIndex , 
	nIndex:= wIndex, 
	pDstBuf:= ADR(aECATParameterReadData), 
	cbBufLen:= SIZEOF(aECATParameterReadData), 
	bExecute:= , 
	tTimeout:= T#1000MS, 
	bCompleteAccess:= FALSE, 
	bBusy=> xBusy, 
	bError=> , 
	nErrId=> , 
	cbRead=> );
	


CASE iStep OF
	0:
	  FOR k:=0 TO 100 DO
		  aECATParameterReadData[k]  := 0;
		  aECATParameterWriteData[k] := 0; 
		  pDestination[k]            := 0;
	  END_FOR;
	  EcCoESdoWriteEx.bExecute := FALSE; 
	  EcCoESdoReadEx.bExecute := FALSE; 
	  istep := istep + 10;
	10:
	   IF R_TRIG_Exec.Q AND xWrite THEN
		   EcCoESdoWriteEx.bExecute := TRUE;
		   xDelayWrite := TRUE;
		   istep := istep + 10;
	   ELSIF R_TRIG_Exec.Q AND NOT xWrite THEN
		   EcCoESdoReadEx.bExecute := TRUE;
		   xDelayRead := TRUE;
		   iStep := 40;
	   END_IF;
	20:
	    IF DelayWrite.Q THEN
			iStep := iStep + 10;
		END_IF;
	
	30:
	    IF NOT EcCoESdoWriteEx.bError THEN
			xDelayWrite := FALSE;
			xDone := TRUE;
			iStep := 60;
	    ELSE
			xError := TRUE;
			xDelayWrite := FALSE;
			udiErrorCode := EcCoESdoWriteEx.nErrId;
			eErrorDescription := TO_DINT(udiErrorCode);
			iStep := 999;
		END_IF;
	40:
	    IF DelayRead.Q THEN
			iStep := iStep + 10;
		END_IF;	
	50:
	    IF NOT EcCoESdoReadEx.bError THEN
			udiReadDataLength := EcCoESdoReadEx.cbRead;
			xDelayRead := FALSE;
			iStep := 60;
	    ELSE
			xError := TRUE;
			xDelayRead := FALSE;
			udiErrorCode := EcCoESdoReadEx.nErrId;
		    eErrorDescription := TO_DINT(udiErrorCode);
			iStep := 999;
		END_IF;	
    60:
	  IF udiReadDataLength >0 THEN
	     xDone := TRUE;
	  END_IF;
	  IF NOT xExecute THEN
		   istep := 0;
	   END_IF;		  	    
	999:
	   IF NOT xExecute THEN
		   istep := 0;
	   END_IF;
	   
	  
END_CASE;

IF F_TRIG_Exec.Q THEN
	iStep :=0;
	xDone := FALSE;
	xBusy := FALSE;
	xError := FALSE;
	udiErrorCode := 0;
    eErrorDescription := 0;
	uiDataLength := 0;
	udiReadDataLength := 0;
END_IF;

END_FUNCTION_BLOCK

// Project Information/F_GetCompany
// This function has been automatically generated from the project information.
{attribute 'signature_flag' := '1073741824'}
{attribute 'TcGenerated'}
{attribute 'no-analysis'}
FUNCTION F_GetCompany : WSTRING
VAR_INPUT
	
END_VAR

F_GetCompany := "Festo";

END_FUNCTION

// Project Information/F_GetTitle
// This function has been automatically generated from the project information.
{attribute 'signature_flag' := '1073741824'}
{attribute 'TcGenerated'}
{attribute 'no-analysis'}
FUNCTION F_GetTitle : WSTRING
VAR_INPUT
	
END_VAR

F_GetTitle := "Festo_CPX_API_EC_Beckhoff";

END_FUNCTION

// Project Information/F_GetVersion
// This function has been automatically generated from the project information.
{attribute 'signature_flag' := '1073741824'}
{attribute 'TcGenerated'}
{attribute 'no-analysis'}
FUNCTION F_GetVersion : ST_LibVersion
VAR_INPUT
	
END_VAR

F_GetVersion.iMajor := 3;
F_GetVersion.iMinor := 5;
F_GetVersion.iBuild := 12;
F_GetVersion.iRevision := 2;

END_FUNCTION

// VISUs/VISU_CPXAPI_Diag
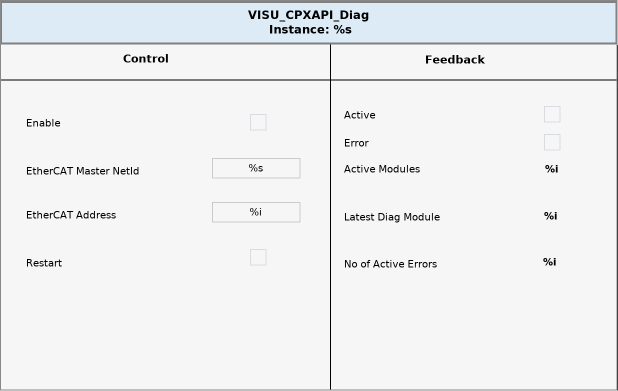
VISUALIZATION VISU_CPXAPI_Diag  // 618x391
{attribute 'hide'}
VAR_INPUT
	{attribute 'parameterstringof' := 'VISU_CPXAPI_Diag'}
	m_Input_INST_str 	: STRING;
END_VAR
VAR_IN_OUT
	VISU_CPXAPI_Diag : CPXAPI_Diag;
END_VAR
    Line (330,42) (330,390)
    Rectangle (0,1 617x43), "VISU_CPXAPI_Diag Instance: %s", text variable: m_Input_INST_str
    Label (116,49 60x20), "Control"
    Label (411,50 88x20), "Feedback"
    Label (23,205 112x20), "EtherCAT Address"
    Rectangle (212,202 88x20), "%i", tooltip "EtherCAT Address of CPX_AP_I_EC_M12.", text variable: VISU_CPXAPI_Diag.uiEthercatAddress
        OnMouseDown: write the text variable via Edit
    Label (23,113 120x20), "Enable"
    Label (341,133 120x20), "Error"
    RoundedRectangle (250,114 16x16), tooltip "Enable Diagnosis", colour toggle: VISU_CPXAPI_Diag.xEnable
        toggle VISU_CPXAPI_Diag.xEnable
    RoundedRectangle (250,249 16x16), tooltip "Restart the EtherCAT Slave devices", colour toggle: VISU_CPXAPI_Diag.xRestart
        toggle VISU_CPXAPI_Diag.xRestart
    RoundedRectangle (544,134 16x16), colour toggle: VISU_CPXAPI_Diag.xError
    Rectangle (493,206 116x20), "%i", text variable: VISU_CPXAPI_Diag.uiModuleNo, colour toggle: VISU_CPXAPI_Diag.uiModuleNo
    Rectangle (492,252 116x20), "%i", text variable: VISU_CPXAPI_Diag.uiNumberOfActiveErrors, colour toggle: VISU_CPXAPI_Diag.uiNumberOfActiveErrors
    Label (341,159 120x20), "Active Modules"
    Label (341,207 120x20), "Latest Diag Module"
    Label (341,254 157x20), "No of Active Errors"
    Label (23,253 112x20), "Restart"
    Line (617,80) (0,80)
    Line (617,45) (617,390)
    Rectangle (494,159 116x20), "%i", text variable: VISU_CPXAPI_Diag.uiActiveModules, colour toggle: VISU_CPXAPI_Diag.uiActiveModules
    Line (617,390) (1,390)
    Label (23,161 123x20), "EtherCAT Master NetId"
    Rectangle (212,158 88x20), "%s", tooltip "EtherCAT Master NetId.", text variable: VISU_CPXAPI_Diag.sNetId
        OnMouseDown: write the text variable via Edit
    Label (341,105 120x20), "Active"
    RoundedRectangle (544,106 16x16), colour toggle: VISU_CPXAPI_Diag.xActive
END_VISUALIZATION

// VISUs/VISU_CPXAPI_IOLinkParameter
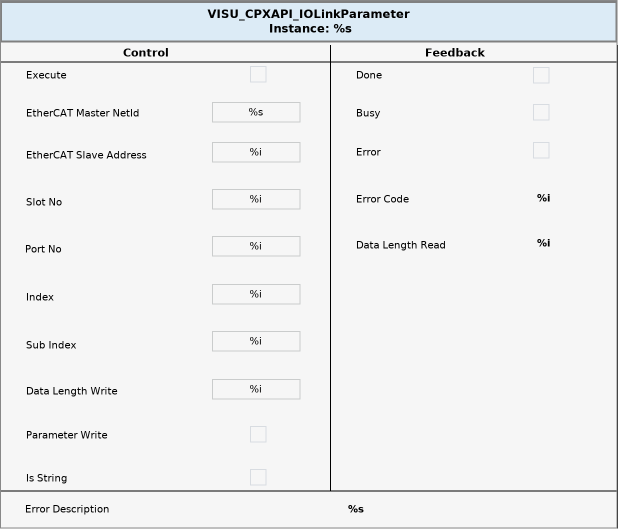
VISUALIZATION VISU_CPXAPI_IOLinkParameter  // 618x529
{attribute 'hide'}
VAR_INPUT
	{attribute 'parameterstringof' := 'VISU_CPXAPI_IOLinkParameter'}
	m_Input_INST_str 	: STRING;
END_VAR
VAR_IN_OUT
	VISU_CPXAPI_IOLinkParameter : CPXAPI_IOLink_Parameter;
END_VAR
    Line (330,45) (330,490)
    Rectangle (0,1 617x41), "VISU_CPXAPI_IOLinkParameter Instance: %s", text variable: m_Input_INST_str
    Label (116,43 60x20), "Control"
    Label (411,43 88x20), "Feedback"
    Label (23,145 131x20), "EtherCAT Slave Address"
    Rectangle (212,142 88x20), "%i", tooltip "EtherCAT Address of CPX-AP-I-EC-M12.", text variable: VISU_CPXAPI_IOLinkParameter.uiEthercatAddress
        OnMouseDown: write the text variable via Edit
    Label (23,65 120x20), "Execute"
    Label (23,425 120x20), "Parameter Write"
    Label (353,65 120x20), "Done"
    Label (353,103 120x20), "Busy"
    Line (617,528) (1,528)
    RoundedRectangle (250,66 16x16), tooltip "Start Parameter Read/Write", colour toggle: VISU_CPXAPI_IOLinkParameter.xExecute
        toggle VISU_CPXAPI_IOLinkParameter.xExecute
    RoundedRectangle (250,426 16x16), tooltip "Execute Parameter Write operation.", colour toggle: VISU_CPXAPI_IOLinkParameter.xReadWrite
        toggle VISU_CPXAPI_IOLinkParameter.xReadWrite
    RoundedRectangle (533,67 16x16), colour toggle: VISU_CPXAPI_IOLinkParameter.xDone
    RoundedRectangle (533,104 16x16), colour toggle: VISU_CPXAPI_IOLinkParameter.xBusy
    RoundedRectangle (533,142 16x16), colour toggle: VISU_CPXAPI_IOLinkParameter.xError
    Rectangle (486,188 116x20), "%i", text variable: VISU_CPXAPI_IOLinkParameter.udiErrorCode
    Rectangle (486,233 116x20), "%i", text variable: VISU_CPXAPI_IOLinkParameter.udiReadDataLength
    Label (353,142 120x20), "Error"
    Label (353,189 120x20), "Error Code"
    Label (353,235 120x20), "Data Length Read"
    Label (23,287 112x20), "Index"
    Label (23,335 112x20), "Sub Index"
    Rectangle (212,284 88x20), "%i", tooltip "Index of the Parameter.", text variable: VISU_CPXAPI_IOLinkParameter.uiIndex
        OnMouseDown: write the text variable via Edit
    Rectangle (212,331 88x20), "%i", tooltip "Sub Index of the parameter.", text variable: VISU_CPXAPI_IOLinkParameter.usiSubIndex
        OnMouseDown: write the text variable via Edit
    Label (23,381 112x20), "Data Length Write"
    Rectangle (212,379 88x20), "%i", tooltip "Length of Data to be written to a parameter.", text variable: VISU_CPXAPI_IOLinkParameter.uiDataLength
        OnMouseDown: write the text variable via Edit
    Line (617,62) (0,62)
    Line (617,45) (617,528)
    Label (23,468 120x20), "Is String"
    RoundedRectangle (250,469 16x16), tooltip "Parameter Data is of STRING Data Type.", colour toggle: VISU_CPXAPI_IOLinkParameter.xIsString
        toggle VISU_CPXAPI_IOLinkParameter.xIsString
    Label (23,192 112x20), "Slot No"
    Label (22,239 112x20), "Port No"
    Rectangle (212,189 88x20), "%i", tooltip "Slot where the CPX-AP-I-4IOL IO Link Master is connected.", text variable: VISU_CPXAPI_IOLinkParameter.uiSlotNumber
        OnMouseDown: write the text variable via Edit
    Rectangle (212,236 88x20), "%i", tooltip "Port of CPX-AP-I-4IOL where the IO Link device is connected", text variable: VISU_CPXAPI_IOLinkParameter.usiPort
        OnMouseDown: write the text variable via Edit
    Line (616,491) (0,491)
    Label (22,499 120x20), "Error Description"
    Rectangle (131,499 450x20), "%s", text variable: VISU_CPXAPI_IOLinkParameter.eErrorDescription
    Label (23,103 123x20), "EtherCAT Master NetId"
    Rectangle (212,102 88x20), "%s", tooltip "EtherCAT Master NetId", text variable: VISU_CPXAPI_IOLinkParameter.sNetId
        OnMouseDown: write the text variable via Edit
END_VISUALIZATION

// VISUs/VISU_CPXAPI_Parameter
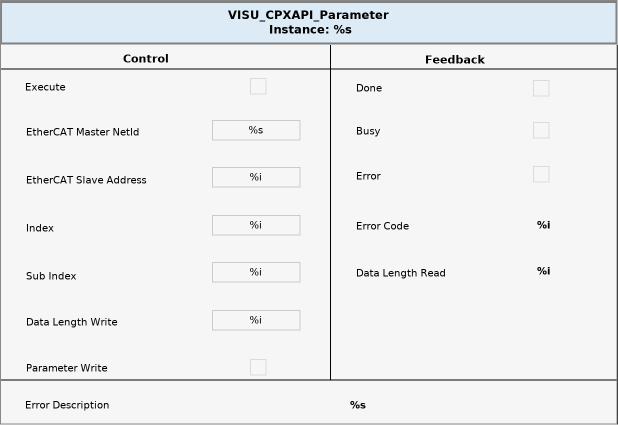
VISUALIZATION VISU_CPXAPI_Parameter  // 618x425
{attribute 'hide'}
VAR_INPUT
	{attribute 'parameterstringof' := 'VISU_CPXAPI_Parameter'}
	m_Input_INST_str 	: STRING;
END_VAR
VAR_IN_OUT
	VISU_CPXAPI_Parameter : CPXAPI_Parameter;
END_VAR
    Line (330,45) (330,380)
    Rectangle (0,1 617x43), "VISU_CPXAPI_Parameter Instance: %s", text variable: m_Input_INST_str
    Label (116,49 60x20), "Control"
    Label (411,50 88x20), "Feedback"
    Label (23,170 133x20), "EtherCAT Slave Address"
    Rectangle (212,167 88x20), "%i", tooltip "EtherCAT Address of CPX-AP-I-EC-M12.", text variable: VISU_CPXAPI_Parameter.uiEthercatAddress
        OnMouseDown: write the text variable via Edit
    Label (23,122 133x20), "EtherCAT Master NetId"
    Label (23,358 120x20), "Parameter Write"
    Label (353,78 120x20), "Done"
    Label (353,121 120x20), "Busy"
    Line (617,424) (1,424)
    RoundedRectangle (250,78 16x16), tooltip "Start Parameter Read/Write", colour toggle: VISU_CPXAPI_Parameter.xExecute
        toggle VISU_CPXAPI_Parameter.xExecute
    RoundedRectangle (250,359 16x16), tooltip "Execute Parameter Write operation.", colour toggle: VISU_CPXAPI_Parameter.xReadWrite
        toggle VISU_CPXAPI_Parameter.xReadWrite
    RoundedRectangle (533,80 16x16), colour toggle: VISU_CPXAPI_Parameter.xDone
    RoundedRectangle (533,122 16x16), colour toggle: VISU_CPXAPI_Parameter.xBusy
    RoundedRectangle (533,166 16x16), colour toggle: VISU_CPXAPI_Parameter.xError
    Rectangle (486,215 116x20), "%i", text variable: VISU_CPXAPI_Parameter.udiErrorCode
    Rectangle (486,261 116x20), "%i", text variable: VISU_CPXAPI_Parameter.udiReadDataLength
    Label (353,166 120x20), "Error"
    Label (353,216 120x20), "Error Code"
    Label (353,263 120x20), "Data Length Read"
    Label (23,218 112x20), "Index"
    Label (23,266 112x20), "Sub Index"
    Rectangle (212,215 88x20), "%i", tooltip "Parameter Index.", text variable: VISU_CPXAPI_Parameter.wIndex
        OnMouseDown: write the text variable via Edit
    Rectangle (212,262 88x20), "%i", tooltip "Parameter Sub Index", text variable: VISU_CPXAPI_Parameter.bySubIndex
        OnMouseDown: write the text variable via Edit
    Label (23,312 112x20), "Data Length Write"
    Rectangle (212,310 88x20), "%i", tooltip "Length of data to be written to a parameter.", text variable: VISU_CPXAPI_Parameter.uiDataLength
        OnMouseDown: write the text variable via Edit
    Line (617,69) (0,69)
    Line (617,45) (617,424)
    Line (617,380) (1,380)
    Label (22,395 120x20), "Error Description"
    Rectangle (133,395 450x20), "%s", text variable: VISU_CPXAPI_Parameter.eErrorDescription
    Label (22,77 120x20), "Execute"
    Rectangle (212,120 88x20), "%s", tooltip "EtherCAT Master NetId.", text variable: VISU_CPXAPI_Parameter.sNetId
        OnMouseDown: write the text variable via Edit
END_VISUALIZATION
